{attribute 'linkalways'} 
{attribute 'no_explicit_call' := 'This FB is a CLASS and must be accessed using methods or properties'}
{attribute 'enable_dynamic_creation'}
FUNCTION_BLOCK Node_F_VN_RotateImage EXTENDS VisionNode
VAR
    ipSrcImage : _ITcVnImage;
    ipDestImage : _ITcVnImage;
    eAngle : _ETcVnRotationAngle(ETcVnRotationAngle.TCVN_RA_90_DEG);
    hrPrev : _HRESULT(S_OK);
	hresult : _HRESULT(S_OK);
END_VAR

METHOD PUBLIC  Clone : I_Node
VAR
	pNode : POINTER TO Node_F_VN_RotateImage;
END_VAR
pNode := __NEW(Node_F_VN_RotateImage);
Clone := pNode^;
END_METHOD

METHOD FB_init : BOOL
VAR_INPUT
	bInitRetains : BOOL; // if TRUE, the retain variables are initialized (warm start / cold start)
	bInCopyCode : BOOL;  // if TRUE, the instance afterwards gets moved into the copy code (online change)
END_VAR
AddInput('ipSrcImage', ipSrcImage);
AddParameter('eAngle', eAngle);
AddInput('hrPrev', hrPrev);
AddOutput('ipDestImage', ipDestImage);
AddOutput('hresult',hresult);
END_METHOD

METHOD PROTECTED OnExecute
hresult.Value := F_VN_RotateImage(
    ipSrcImage := ipSrcImage.Value,
	ipDestImage := ipDestImage.Value,
    eAngle := eAngle.Value,
	hrPrev:= hrPrev.Value);
END_METHOD

METHOD PUBLIC PreExecutionCheck
VAR_INPUT
	Check : I_PreExecutionChecks;
END_VAR
Check.IsTrue(ipSrcImage.IsValid, 'ipSrcImage must contain an image');
END_METHOD

END_FUNCTION_BLOCK

(* stored: Version 1.1.0.1, ProductVersion 3.1.4024.13
   POU Node_F_VN_RotateImage: Id {d65f53e6-8171-0e7e-09ba-3559a68a008a}, SpecialFunc None
   Folder Constructor: Id {c8fca73b-ca2e-0a09-1aa7-58201e9ee224}
   Method Clone: Id {2b6b52b9-efcc-0ade-3fd7-3d829ce1c9d3}
   Method FB_init: Id {1b183d22-a404-06a3-1b30-ba371900a898}
   Method OnExecute: Id {d40f3c52-106a-021a-2edf-741b56fc7924}
   Method PreExecutionCheck: Id {34d181aa-fdec-068a-3e9d-6b8fb28dfc1a} *)
